FUNCTION_BLOCK LED
VAR
	bOutputActive AT %I*: BOOL;
	bOutputSetpoint AT %Q*: BOOL;
	nCurrent AT %I*: UINT;
	nOutputCurrent: UINT;
END_VAR

IF bOutputActive THEN
	nOutputCurrent := nCurrent;
ELSE
	nOutputCurrent := 0;
END_IF

END_FUNCTION_BLOCK

(* stored: Version 1.1.0.1, ProductVersion 3.1.4024.12
   POU LED: Id {6ce5d4a1-e171-47ff-a2a3-978987a72d98}, SpecialFunc None *)
